PROGRAM Main
VAR
	{attribute 'pytmc' := '
        pv: TST:PPM:MMS:Y
	'}
	M1: DUT_MotionStage;
	
	{attribute 'pytmc' := '
		pv: TST
	'}
	fbPPM: FB_PPM;
END_VAR

fbPPM(stYStage := M1);

END_PROGRAM

(* stored: Version 1.1.0.1, ProductVersion 3.1.4020.14
   POU Main: Id {cb921465-efa3-4bda-880b-e8f57acf61aa}, SpecialFunc None *)
